(*
SPDX-FileCopyrightText: © 2026 Oleksandr Tiutyk <trofimich@gmail.com>
SPDX-License-Identifier: MIT
License: https://opensource.org/license/mit
*)

(*!
<summary>Marker interface for a condition that always evaluates to TRUE.</summary>
*)

INTERFACE ITrueCondition EXTENDS ICondition

END_INTERFACE

(* stored: Version 1.1.0.1
   Itf ITrueCondition: Id {cff04628-cc2a-462f-923d-5cefd5145029} *)
